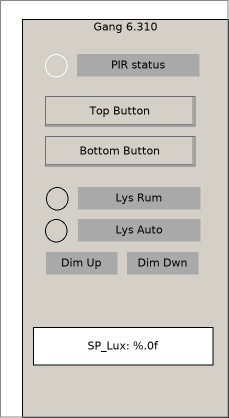
VISUALIZATION Visualization_6_310  // 229x418
    RoundedRectangle (22,19 207x399), "Gang 6.310"
    Rectangle (33,327 180x38), "SP_Lux: %.0f", text variable: P_Gang_6_310.fbLys.fbLightCtrl.fLuxZone1
    Button (45,96 150x30), "Top Button"
        tap P_Gang_6_310.bTopButtonZone1
    Button (45,136 150x30), "Bottom Button"
        tap P_Gang_6_310.bBottomButtonZone1_Visu
    Ellipse (46,187 22x23), colour toggle: P_Gang_6_310.fbLys.fbLightCtrl.bOnZone1
    Rectangle (78,187 122x22), "Lys Rum"
    Rectangle (46,252 71x22), "Dim Up", colour toggle: P_Gang_6_310.fbLys.fbLightCtrl.bDimUp
    Rectangle (127,252 71x22), "Dim Dwn", colour toggle: P_Gang_6_310.fbLys.fbLightCtrl.bDimDwn
    Ellipse (45,219 22x23), colour toggle: P_Gang_6_310.fbLys.fbLightCtrl.bAutoZone1
    Rectangle (78,219 122x22), "Lys Auto"
    Ellipse (45,54 22x23), colour toggle: P_Gang_6_310.fbLys.fbLightCtrl.bPIR
    Rectangle (77,54 122x22), "PIR status"
END_VISUALIZATION

(* stored: Version 1.1.0.1
   Visu Visualization_6_310: Id {b34e3b65-7d4e-4356-b2a4-9c40488202f7} *)
